VAR_GLOBAL

END_VAR

(* stored: Version 1.1.0.1, ProductVersion 3.1.4018.5
   GVL GVL_Simulations_Haus: Id {e6ed5590-eeb1-43b7-b0d3-ec7308a276ec} *)
